FUNCTION AddRequest : BOOL
VAR_INPUT
	
END_VAR
VAR
END_VAR
VAR_OUTPUT
	bFinishStatus: BOOL;
END_VAR

END_FUNCTION

(* stored: Version 1.1.0.1, ProductVersion 3.1.4022.12
   POU AddRequest: Id {8eefe877-badb-46e8-adb3-f23ae5cd2f81}, SpecialFunc None *)
